(* IEC 61131-3 sources: Industry-PLC-LLM/data/PLCBEAD_repo/PLCBEAD_PLCEmbed-main/PLC-BEAD/Source/GEB/ERFC, 1 file *)

(* ---- ERFC.ST ---- *)
FUNCTION SGN : INT
  VAR_INPUT
    X : REAL;
  END_VAR

  IF X > 0.0 THEN
  	SGN := 1;
  ELSIF X < 0.0 THEN
  	SGN := -1;
  ELSE
  	SGN := 0;
  END_IF;
END_FUNCTION

FUNCTION ERF:REAL

	VAR_INPUT
		X :	REAL;
	END_VAR

	VAR
		X2 :	REAL;
		AX2 :	REAL;
	END_VAR

	X2 := X*X;
	AX2 := 0.147 * X2 + 1.0;
	ERF := SQRT(1.0 - EXP(-X2 * ((0.27323954473516 + AX2)/(AX2)))) * INT_TO_REAL(SGN(X));

END_FUNCTION

FUNCTION ERFC:REAL
	VAR_INPUT
		X :	REAL;
	END_VAR

	ERFC := 1.0 - ERF(X);

END_FUNCTION

PROGRAM program0
  VAR
    LocalVar0 : REAL;
	  LocalOUT  : REAL;
  END_VAR
  	LocalOUT := ERFC(LocalVar0);
END_PROGRAM
